// TIA Portal V20 export
FUNCTION_BLOCK "Com"   // FB301, FBD
{ S7_Optimized_Access := 'FALSE' }
// stored: AutoNumber false, SetENOAutomatically false
   VAR
      Var { S7_SetPoint := 'True'} : "TypeVar";
      T : Array[1..6] of IEC_TIMER;
      wdOldParam { ExternalAccessible := 'False'; ExternalVisible := 'False'; ExternalWritable := 'False'} : Int;
      wdOldErr { ExternalAccessible := 'False'; ExternalVisible := 'False'; ExternalWritable := 'False'} : Int;
   END_VAR
   VAR_TEMP   // added for the SCL form of the ladder/FBD networks
      _w1 : Bool;
   END_VAR
BEGIN

REGION Network 1 (SCL): version info
   "ComSd".Data.config.Version := 13;

   IF "ComRd".Data.Config.version <> "ComSd".Data.config.Version THEN
       "G".errVersion := TRUE;
   ELSE
       "G".errVersion := FALSE;
   END_IF;

   IF "G".ack THEN
       "G".errVersion := FALSE;
   END_IF;
END_REGION

REGION Network 2: valid
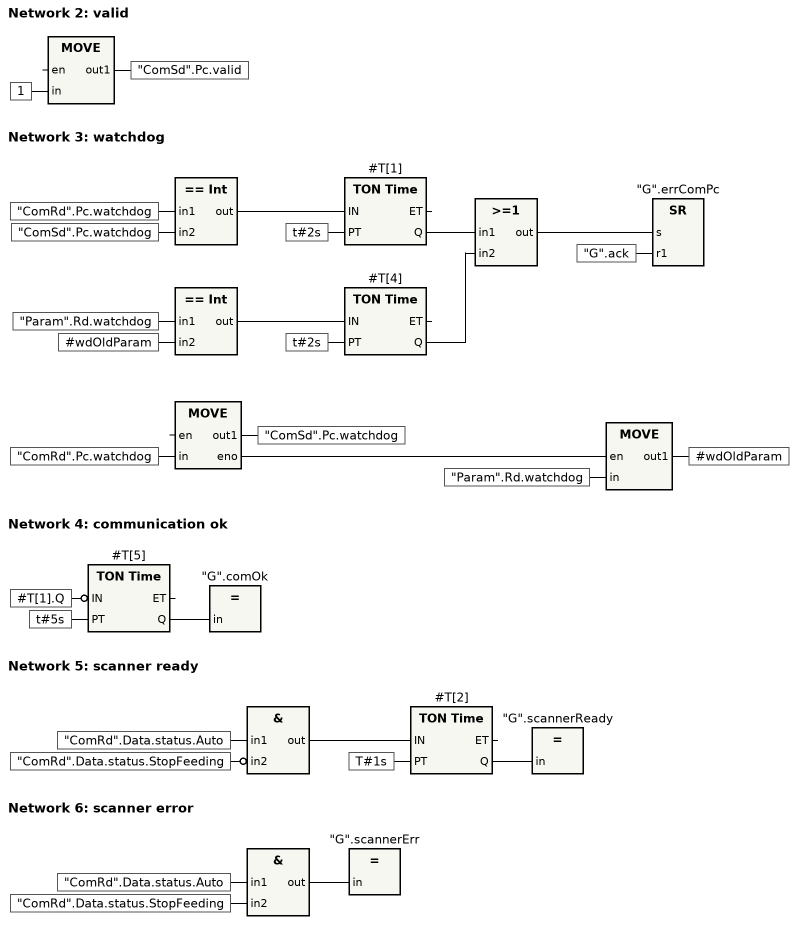
   "ComSd".Pc.valid := 1;
END_REGION

REGION Network 3: watchdog
   #T[1].TON(IN := "ComRd".Pc.watchdog = "ComSd".Pc.watchdog, PT := t#2s);
   #_w1 := #T[1].Q;
   #T[4].TON(IN := "Param".Rd.watchdog = #wdOldParam, PT := t#2s);
   IF #_w1 OR #T[4].Q THEN
       "G".errComPc := TRUE;   // SR flip-flop
   END_IF;
   IF "G".ack THEN "G".errComPc := FALSE; END_IF;
   "ComSd".Pc.watchdog := "ComRd".Pc.watchdog;
   #wdOldParam := "Param".Rd.watchdog;
END_REGION

REGION Network 4: communication ok
   #T[5].TON(IN := NOT #T[1].Q, PT := t#5s);
   "G".comOk := #T[5].Q;
END_REGION

REGION Network 5: scanner ready
   #T[2].TON(IN := "ComRd".Data.status.Auto AND NOT "ComRd".Data.status.StopFeeding, PT := T#1s);
   "G".scannerReady := #T[2].Q;
END_REGION

REGION Network 6: scanner error
   "G".scannerErr := "ComRd".Data.status.Auto AND "ComRd".Data.status.StopFeeding;
END_REGION

REGION Network 7: release infeed
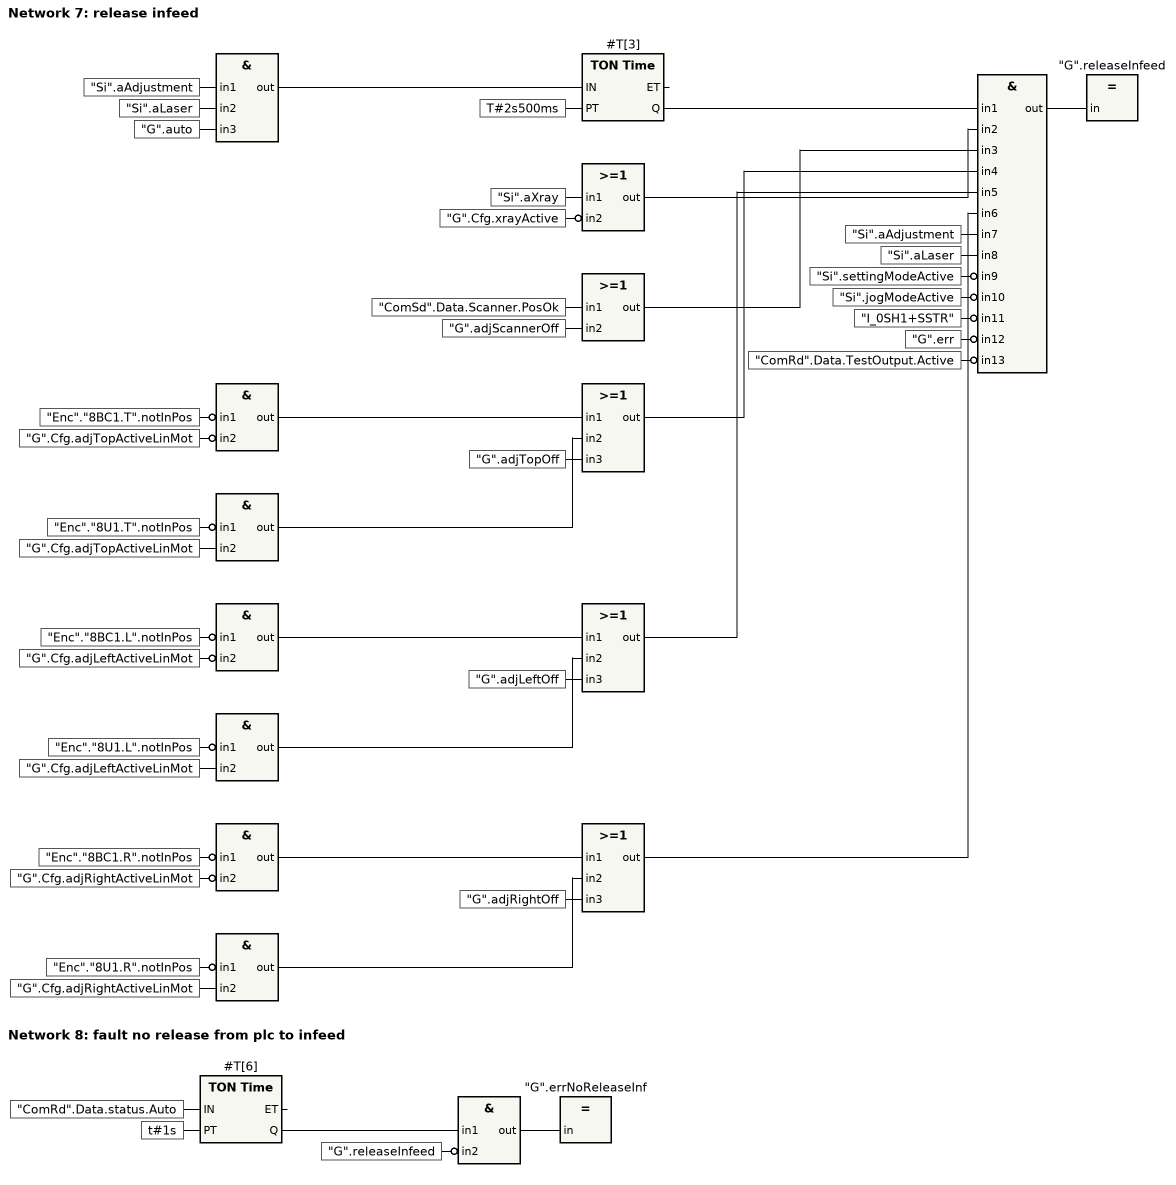
   #T[3].TON(IN := "Si".aAdjustment AND "Si".aLaser AND "G".auto, PT := T#2s500ms);
   "G".releaseInfeed := #T[3].Q AND ("Si".aXray OR NOT "G".Cfg.xrayActive) AND ("ComSd".Data.Scanner.PosOk OR "G".adjScannerOff) AND ((NOT "Enc"."8BC1.T".notInPos AND NOT "G".Cfg.adjTopActiveLinMot) OR (NOT "Enc"."8U1.T".notInPos AND "G".Cfg.adjTopActiveLinMot) OR "G".adjTopOff) AND ((NOT "Enc"."8BC1.L".notInPos AND NOT "G".Cfg.adjLeftActiveLinMot) OR (NOT "Enc"."8U1.L".notInPos AND "G".Cfg.adjLeftActiveLinMot) OR "G".adjLeftOff) AND ((NOT "Enc"."8BC1.R".notInPos AND NOT "G".Cfg.adjRightActiveLinMot) OR (NOT "Enc"."8U1.R".notInPos AND "G".Cfg.adjRightActiveLinMot) OR "G".adjRightOff) AND "Si".aAdjustment AND "Si".aLaser AND NOT "Si".settingModeActive AND NOT "Si".jogModeActive AND NOT "I_0SH1+SSTR" AND NOT "G".err AND NOT "ComRd".Data.TestOutput.Active;
END_REGION

REGION Network 8: fault no release from plc to infeed
   #T[6].TON(IN := "ComRd".Data.status.Auto, PT := t#1s);
   "G".errNoReleaseInf := #T[6].Q AND NOT "G".releaseInfeed;
END_REGION

REGION Network 9: communication signals
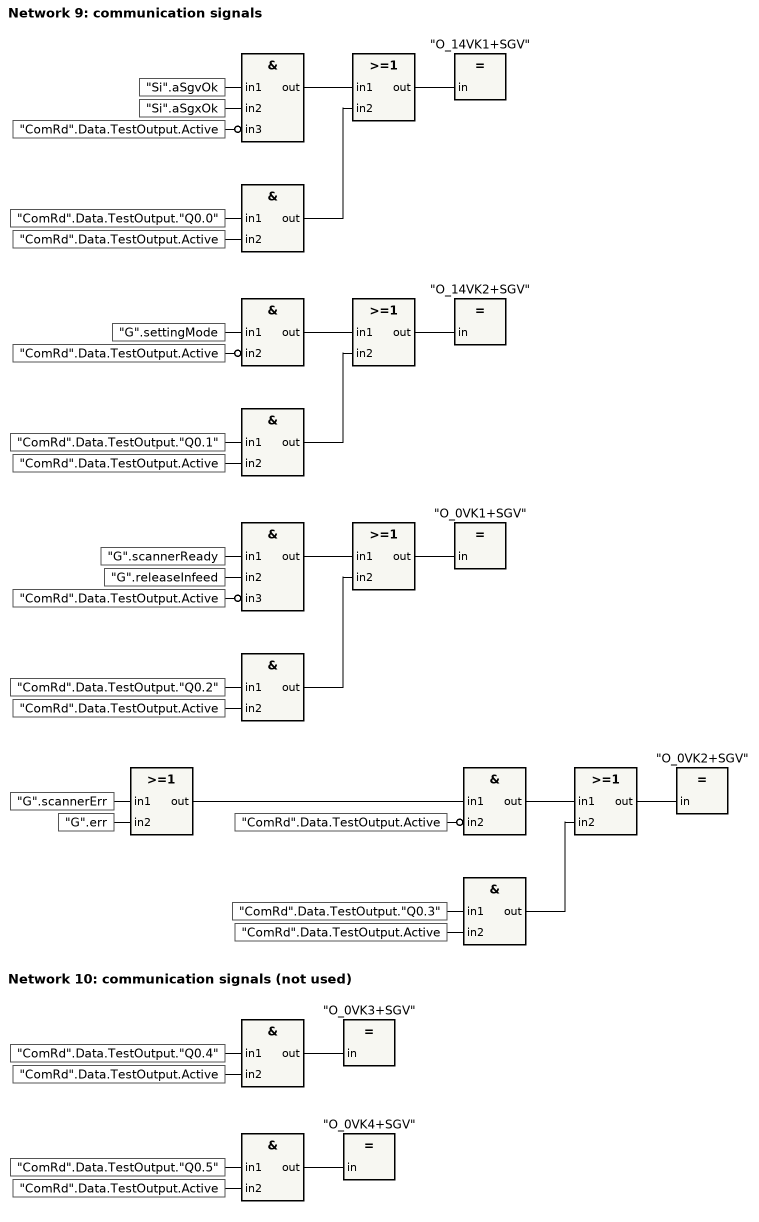
   "O_14VK1+SGV" := ("Si".aSgvOk AND "Si".aSgxOk AND NOT "ComRd".Data.TestOutput.Active) OR ("ComRd".Data.TestOutput."Q0.0" AND "ComRd".Data.TestOutput.Active);
   "O_14VK2+SGV" := ("G".settingMode AND NOT "ComRd".Data.TestOutput.Active) OR ("ComRd".Data.TestOutput."Q0.1" AND "ComRd".Data.TestOutput.Active);
   "O_0VK1+SGV" := ("G".scannerReady AND "G".releaseInfeed AND NOT "ComRd".Data.TestOutput.Active) OR ("ComRd".Data.TestOutput."Q0.2" AND "ComRd".Data.TestOutput.Active);
   "O_0VK2+SGV" := (("G".scannerErr OR "G".err) AND NOT "ComRd".Data.TestOutput.Active) OR ("ComRd".Data.TestOutput."Q0.3" AND "ComRd".Data.TestOutput.Active);
END_REGION

REGION Network 10: communication signals (not used)
   "O_0VK3+SGV" := "ComRd".Data.TestOutput."Q0.4" AND "ComRd".Data.TestOutput.Active;
   "O_0VK4+SGV" := "ComRd".Data.TestOutput."Q0.5" AND "ComRd".Data.TestOutput.Active;
END_REGION

REGION Network 11 (SCL): send
   // data - safety
   "ComSd".Data.safety.AreaAdjustmentOn := "Si".aAdjustment;
   "ComSd".Data.safety.AreaLaserOn := "Si".aLaser;
   "ComSd".Data.safety.AreaXrayOn := "Si".aXray;

   // data - status
   "ComSd".Data.status.err := "G".err;
   "ComSd".Data.status.ready := "G".scannerReady AND "G".releaseInfeed;
END_REGION
END_FUNCTION_BLOCK
